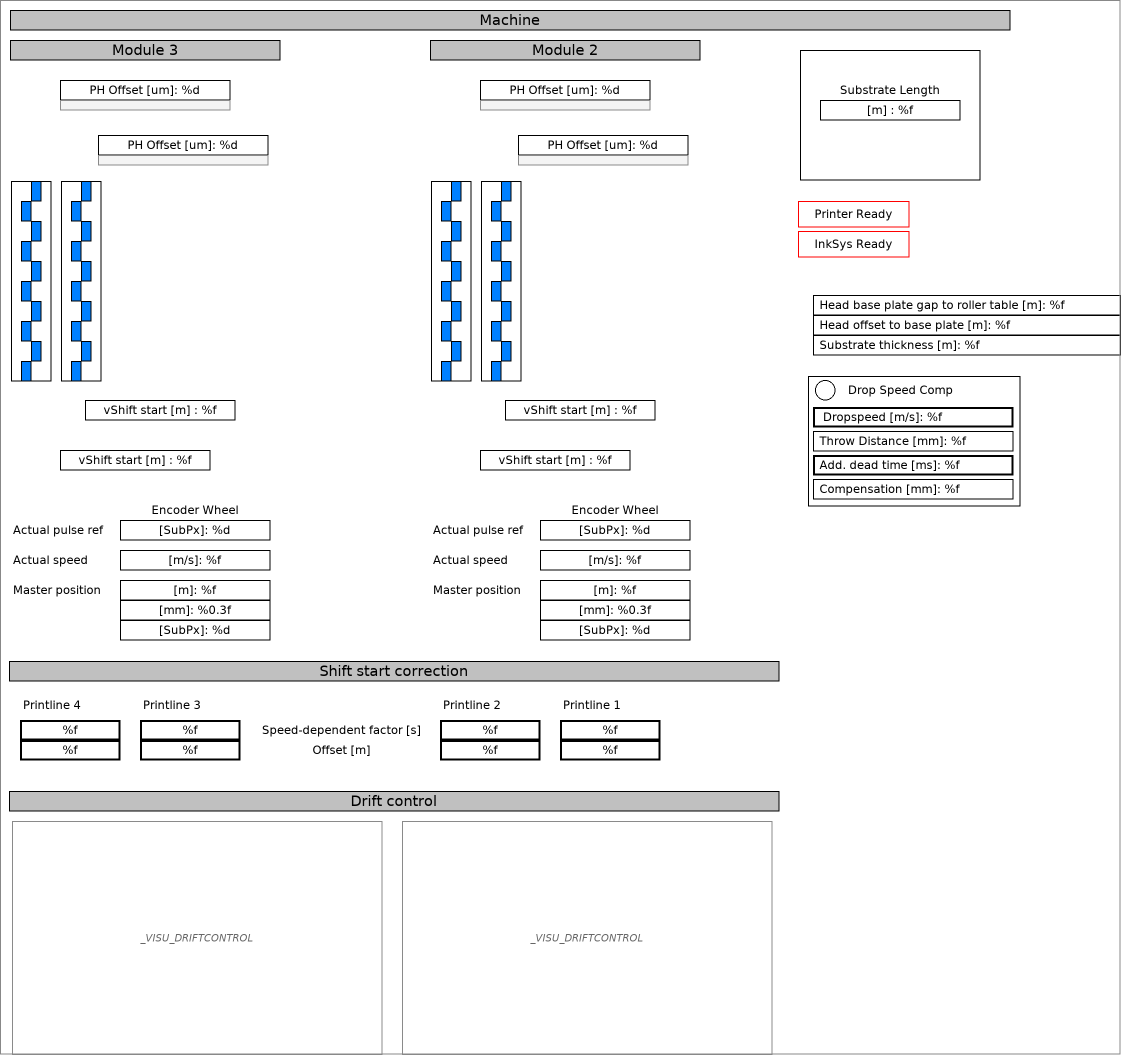
VISUALIZATION VISU_PAPER_POS_DETECT  // 1121x1055
    Polyline (100,340)
    Rectangle (800,50 180x130)
    Rectangle (10,10 1000x20), "Machine"
    Rectangle (820,100 140x20), "[m] : %f", text variable: PRG_PRINT.fL_SubstrateLen[ePr_PG_GROUP_1]
        OnMouseDown: write the text variable via Edit
    Rectangle (820,80 140x20), "Substrate Length"
    Rectangle (798,201 111x26), "Printer Ready", colour toggle: PRG_MACHINE.bO_PrinterReady
    Rectangle (798,231 111x26), "InkSys Ready", colour toggle: PRG_INK.bO_InkSystemOk
    Rectangle (808,376 212x130)
    Ellipse (815,380 20x20), colour toggle: PRG_PRINT.bL_UseSpeedCompensation
        toggle PRG_PRINT.bL_UseSpeedCompensation
    Rectangle (845,380 124x20), "Drop Speed Comp"
    Rectangle (813,407 200x20), "Dropspeed [m/s]: %f", text variable: PRG_PRINT.fL_DropSpeed
        OnMouseDown: write the text variable via Edit
    Rectangle (813,431 200x20), "Throw Distance [mm]: %f", text variable: PRG_PRINT.fL_PrintUnitElevation[1]
    Rectangle (813,479 200x20), "Compensation [mm]: %f", text variable: 1000 * PRG_PRINT.fL_SpeedComp[ePr_PU_UNIT_1]
    Rectangle (813,455 200x20), "Add. dead time [ms]: %f", text variable: PRG_PRINT.fL_DropSpeedAddTime
        OnMouseDown: write the text variable via Edit
    Rectangle (813,295 308x20), "Head base plate gap to roller table [m]: %f", text variable: PRG_PRINT.fL_HeadGap[1], invisible if: TRUE
        OnMouseDown: write the text variable via Edit
    Rectangle (813,315 308x20), "Head offset to base plate [m]: %f", text variable: PRG_PRINT.fL_HeadOffsetPlate, invisible if: TRUE
        OnMouseDown: write the text variable via Edit
    Rectangle (813,335 308x20), "Substrate thickness [m]: %f", text variable: PRG_PRINT.fL_SubstrateThickness, invisible if: TRUE
        OnMouseDown: write the text variable via Edit
    Group (61,181 38x198)
        Rectangle (0,0 40x200)
        Rectangle (20,0 10x20)
        Rectangle (10,20 10x20)
        Rectangle (20,40 10x20)
        Rectangle (10,60 10x20)
        Rectangle (20,80 10x20)
        Rectangle (10,100 10x20)
        Rectangle (20,120 10x20)
        Rectangle (10,140 10x20)
        Rectangle (20,160 10x20)
        Rectangle (10,180 10x20)
    Group (11,181 38x198)
        Rectangle (0,0 40x200)
        Rectangle (20,0 10x20)
        Rectangle (10,20 10x20)
        Rectangle (20,40 10x20)
        Rectangle (10,60 10x20)
        Rectangle (20,80 10x20)
        Rectangle (10,100 10x20)
        Rectangle (20,120 10x20)
        Rectangle (10,140 10x20)
        Rectangle (20,160 10x20)
        Rectangle (10,180 10x20)
    Rectangle (60,80 170x20), "PH Offset [um]: %d", text variable: PRG_PRINT.sAdsPrintGroup[ePr_PG_GROUP_4].sI_ShiftPositionX.lI_Val
        OnMouseDown: write the text variable via Edit
    Scrollbar (60,100 170x10)
        p1057716461: PRG_PRINT.sAdsPrintGroup[ePr_PG_GROUP_2].sI_ShiftPositionX.lI_Val
    Polyline (100,140)
    Polyline (150,360)
    Rectangle (98,135 170x20), "PH Offset [um]: %d", text variable: PRG_PRINT.sAdsPrintGroup[ePr_PG_GROUP_3].sI_ShiftPositionX.lI_Val
        OnMouseDown: write the text variable via Edit
    Scrollbar (98,155 170x10)
        p1057716461: PRG_PRINT.sAdsPrintGroup[ePr_PG_GROUP_1].sI_ShiftPositionX.lI_Val
    Polyline (150,360)
    Polyline (250,350)
    Rectangle (85,400 150x20), "vShift start [m] : %f", text variable: PRG_PRINT.fbWorkerWeu[3].fPosition
    Rectangle (60,450 150x20), "vShift start [m] : %f", text variable: PRG_PRINT.fbWorkerWeu[4].fPosition
    Polyline (100,340)
    Group (481,181 38x198)
        Rectangle (0,0 40x200)
        Rectangle (20,0 10x20)
        Rectangle (10,20 10x20)
        Rectangle (20,40 10x20)
        Rectangle (10,60 10x20)
        Rectangle (20,80 10x20)
        Rectangle (10,100 10x20)
        Rectangle (20,120 10x20)
        Rectangle (10,140 10x20)
        Rectangle (20,160 10x20)
        Rectangle (10,180 10x20)
    Group (431,181 38x198)
        Rectangle (0,0 40x200)
        Rectangle (20,0 10x20)
        Rectangle (10,20 10x20)
        Rectangle (20,40 10x20)
        Rectangle (10,60 10x20)
        Rectangle (20,80 10x20)
        Rectangle (10,100 10x20)
        Rectangle (20,120 10x20)
        Rectangle (10,140 10x20)
        Rectangle (20,160 10x20)
        Rectangle (10,180 10x20)
    Rectangle (480,80 170x20), "PH Offset [um]: %d", text variable: PRG_PRINT.sAdsPrintGroup[ePr_PG_GROUP_2].sI_ShiftPositionX.lI_Val
        OnMouseDown: write the text variable via Edit
    Scrollbar (480,100 170x10)
        p1057716461: PRG_PRINT.sAdsPrintGroup[ePr_PG_GROUP_2].sI_ShiftPositionX.lI_Val
    Polyline (100,140)
    Polyline (150,360)
    Rectangle (518,135 170x20), "PH Offset [um]: %d", text variable: PRG_PRINT.sAdsPrintGroup[ePr_PG_GROUP_1].sI_ShiftPositionX.lI_Val
        OnMouseDown: write the text variable via Edit
    Scrollbar (518,155 170x10)
        p1057716461: PRG_PRINT.sAdsPrintGroup[ePr_PG_GROUP_1].sI_ShiftPositionX.lI_Val
    Polyline (150,360)
    Polyline (250,350)
    Rectangle (505,400 150x20), "vShift start [m] : %f", text variable: PRG_PRINT.fbWorkerWeu[1].fPosition
    Rectangle (480,450 150x20), "vShift start [m] : %f", text variable: PRG_PRINT.fbWorkerWeu[2].fPosition
    Rectangle (10,40 270x20), "Module 3"
    Rectangle (430,40 270x20), "Module 2"
    Rectangle (120,600 150x20), "[mm]: %0.3f", text variable: 0.001*PRG_PRINT.Fb_Ph_Master[ePr_PG_GROUP_2].fO_Master_Position
    Rectangle (120,620 150x20), "[SubPx]: %d", text variable: PRG_PRINT.Fb_Ph_Master[ePr_PG_GROUP_2].lO_Master_Position
    Rectangle (120,550 150x20), "[m/s]: %f", text variable: PRG_PRINT.Fb_Ph_Master[ePr_PG_GROUP_2].fO_Master_Speed
    Rectangle (10,550 100x20), "Actual speed"
    Rectangle (10,580 100x20), "Master position"
    Rectangle (120,520 150x20), "[SubPx]: %d", text variable: PRG_PRINT.Fb_Ph_Master[ePr_PG_GROUP_2].lI_Reference
    Rectangle (10,520 100x20), "Actual pulse ref"
    Rectangle (120,500 150x20), "Encoder Wheel"
    Rectangle (120,580 150x20), "[m]: %f", text variable: 0.000001*PRG_PRINT.Fb_Ph_Master[ePr_PG_GROUP_2].fO_Master_Position
    Rectangle (540,600 150x20), "[mm]: %0.3f", text variable: 0.001*PRG_PRINT.Fb_Ph_Master[ePr_PG_GROUP_1].fO_Master_Position
    Rectangle (540,620 150x20), "[SubPx]: %d", text variable: PRG_PRINT.Fb_Ph_Master[ePr_PG_GROUP_1].lO_Master_Position
    Rectangle (540,550 150x20), "[m/s]: %f", text variable: PRG_PRINT.Fb_Ph_Master[ePr_PG_GROUP_1].fO_Master_Speed
    Rectangle (430,550 100x20), "Actual speed"
    Rectangle (430,580 100x20), "Master position"
    Rectangle (540,520 150x20), "[SubPx]: %d", text variable: PRG_PRINT.Fb_Ph_Master[ePr_PG_GROUP_1].lI_Reference
    Rectangle (430,520 100x20), "Actual pulse ref"
    Rectangle (540,500 150x20), "Encoder Wheel"
    Rectangle (540,580 150x20), "[m]: %f", text variable: 0.000001*PRG_PRINT.Fb_Ph_Master[ePr_PG_GROUP_1].fO_Master_Position
    Frame (12,821 370x234)
        shows _VISU_DRIFTCONTROL(mRef := PRG_PRINT.fB_DriftControl[2])
    Rectangle (9,791 770x20), "Drift control"
    Frame (402,821 370x234)
        shows _VISU_DRIFTCONTROL(mRef := PRG_PRINT.fB_DriftControl[1])
    Rectangle (9,661 770x20), "Shift start correction"
    Rectangle (560,695 100x20), "Printline 1"
    Rectangle (560,720 100x20), "%f", text variable: PRG_PRINT.fbWorkerWeu[1]._fStartShiftFactor
        OnMouseDown: write the text variable via Edit
    Rectangle (560,740 100x20), "%f", text variable: PRG_PRINT.fbWorkerWeu[1]._fStartShiftOffset
        OnMouseDown: write the text variable via Edit
    Rectangle (250,720 180x20), "Speed-dependent factor [s]"
    Rectangle (250,740 180x20), "Offset [m]"
    Rectangle (440,695 100x20), "Printline 2"
    Rectangle (440,720 100x20), "%f", text variable: PRG_PRINT.fbWorkerWeu[2]._fStartShiftFactor
        OnMouseDown: write the text variable via Edit
    Rectangle (440,740 100x20), "%f", text variable: PRG_PRINT.fbWorkerWeu[2]._fStartShiftOffset
        OnMouseDown: write the text variable via Edit
    Rectangle (140,695 100x20), "Printline 3"
    Rectangle (140,720 100x20), "%f", text variable: PRG_PRINT.fbWorkerWeu[3]._fStartShiftFactor
        OnMouseDown: write the text variable via Edit
    Rectangle (140,740 100x20), "%f", text variable: PRG_PRINT.fbWorkerWeu[3]._fStartShiftOffset
        OnMouseDown: write the text variable via Edit
    Rectangle (20,695 100x20), "Printline 4"
    Rectangle (20,720 100x20), "%f", text variable: PRG_PRINT.fbWorkerWeu[4]._fStartShiftFactor
        OnMouseDown: write the text variable via Edit
    Rectangle (20,740 100x20), "%f", text variable: PRG_PRINT.fbWorkerWeu[4]._fStartShiftOffset
        OnMouseDown: write the text variable via Edit
END_VISUALIZATION

(* stored: Version 1.1.0.1, ProductVersion 3.1.4024.9
   Visu VISU_PAPER_POS_DETECT: Id {460bf862-2228-413c-95ff-5f9712d48677} *)
